Yaskawa INFORM job: X2_55A(90,180).JBI

/JOB
//NAME X2_55A(90,180)
//POS
///NPOS 356,356,356,16,0,0
///TOOL 0
///POSTYPE PULSE
///PULSE
C00000=-1668,-120197,-100216,-7,84052,41
C00001=57589,-42382,-44231,37759,86719,-54272
C00002=65855,-25584,-33137,36767,84603,-51533
C00003=68819,-25314,-30615,36422,82198,-51104
C00004=70004,-25113,-29538,36287,81242,-50929
C00005=71107,-26982,-30843,36133,80649,-50666
C00006=70797,-26613,-30828,36166,80927,-50703
C00007=70799,-26325,-28960,36248,80110,-50973
C00008=70711,-26240,-29288,36240,80345,-50932
C00009=71628,-24021,-27732,36086,80108,-50627
C00010=70711,-26240,-29288,36240,80345,-50932
C00011=69517,-26484,-30393,36372,81303,-51111
C00012=66526,-26862,-32992,36707,83713,-51552
C00013=67184,-38422,-41454,21825,57357,-56847
C00014=69536,-35116,-36433,20931,55446,-56242
C00015=70451,-33735,-34368,20579,54688,-56001
C00016=70453,-33369,-32455,20825,53760,-56193
C00017=71285,-32850,-32302,20328,53712,-55835
C00018=71877,-32425,-32021,19993,53611,-55596
C00019=70458,-33427,-32681,20795,53862,-56169
C00020=69543,-34832,-34766,21144,54620,-56412
C00021=67191,-38201,-39835,22030,56533,-57020
C00022=54852,-62445,-55541,26402,56356,-60471
C00023=66049,-20273,-10630,37753,75560,-54572
C00024=69005,-19201,-7438,37708,73136,-54154
C00025=70188,-18683,-6088,37693,72169,-53986
C00026=71287,-20467,-7387,37603,71596,-53710
C00027=70964,-19947,-7085,37622,71802,-53778
C00028=70966,-19095,-4730,37816,70991,-54071
C00029=70796,-19587,-5250,37820,71120,-54100
C00030=71712,-17458,-3693,37701,70830,-53802
C00031=70796,-19587,-5250,37820,71120,-54100
C00032=66612,-21337,-9914,37854,74525,-54698
C00033=67375,-34871,-26422,23789,50429,-58369
C00034=69718,-31047,-20945,22976,48471,-57749
C00035=70629,-29456,-18687,22656,47689,-57504
C00036=70631,-28720,-16473,23004,46778,-57736
C00037=70516,-28887,-16788,23031,46910,-57759
C00038=71933,-27925,-16136,22175,46608,-57138
C00039=70516,-28887,-16788,23031,46910,-57759
C00040=67258,-34379,-24600,24142,49668,-58622
C00041=57576,-53152,-36186,27516,49078,-61266
C00042=66086,-20118,-10544,37746,75565,-54554
C00043=69039,-19046,-7350,37700,73143,-54137
C00044=70219,-18527,-6000,37685,72176,-53969
C00045=71318,-20312,-7301,37595,71604,-53693
C00046=74451,-19008,-9811,31488,73352,-51630
C00047=71045,-18968,-4611,37811,70952,-54051
C00048=70901,-19378,-5096,37807,71084,-54066
C00049=71814,-17244,-3534,37689,70794,-53769
C00050=70901,-19378,-5096,37807,71084,-54066
C00051=66723,-21136,-9768,37841,74486,-54664
C00052=67447,-34663,-26265,23746,50418,-58339
C00053=69784,-30837,-20782,22936,48460,-57720
C00054=70694,-29244,-18522,22618,47678,-57477
C00055=70696,-28510,-16308,22965,46767,-57708
C00056=70662,-28628,-16633,22933,46904,-57689
C00057=72075,-27660,-15975,22080,46604,-57068
C00058=70662,-28628,-16633,22933,46904,-57689
C00059=67414,-34127,-24457,24044,49660,-58550
C00060=58044,-52471,-35805,27235,49028,-61049
C00061=66074,-20265,-10583,37755,75529,-54572
C00062=69030,-19190,-7387,37710,73105,-54154
C00063=70213,-18669,-6036,37695,72138,-53986
C00064=71313,-20454,-7335,37605,71565,-53710
C00065=76162,-7525,-3808,27332,81993,-47754
C00066=80041,-11320,-7163,21944,78815,-47604
C00067=72377,-20867,-8485,35073,70629,-54310
C00068=73758,-17101,-5731,34844,70264,-53838
C00069=70643,-18935,-5429,37748,71542,-54012
C00070=66856,-20964,-9691,37824,74460,-54615
C00071=67489,-34539,-26167,23723,50410,-58320
C00072=69824,-30709,-20681,22912,48451,-57703
C00073=70732,-29117,-18420,22594,47670,-57460
C00074=70735,-28382,-16205,22941,46757,-57691
C00075=70742,-28505,-16565,22880,46902,-57650
C00076=72154,-27535,-15905,22025,46603,-57029
C00077=70742,-28505,-16565,22880,46902,-57650
C00078=67499,-34008,-24394,23990,49655,-58510
C00079=55453,-57012,-39392,28557,49780,-62094
C00080=66203,-19744,-10147,37744,75471,-54537
C00081=69149,-18659,-6941,37699,73052,-54122
C00082=75064,-17968,-9396,29448,73085,-51466
C00083=75064,-17451,-7778,29552,72447,-51636
C00084=75064,-17968,-9396,29448,73085,-51466
C00085=75946,-19134,-10253,29336,72713,-51212
C00086=75064,-17968,-9396,29448,73085,-51466
C00087=75754,-15898,-7859,29336,72947,-51227
C00088=76424,-13822,-6293,29228,72804,-50997
C00089=75754,-15898,-7859,29336,72947,-51227
C00090=66920,-20695,-9518,37813,74457,-54589
C00091=67621,-34252,-25984,23640,50405,-58260
C00092=69948,-30420,-20490,22831,48447,-57645
C00093=70853,-28824,-18225,22514,47664,-57402
C00094=70856,-28091,-16012,22860,46751,-57633
C00095=70871,-28224,-16368,22798,46887,-57590
C00096=72279,-27249,-15703,21944,46591,-56971
C00097=70871,-28224,-16368,22798,46887,-57590
C00098=67638,-33734,-24209,23906,49640,-58448
C00099=55815,-56530,-39132,28348,49735,-61930
C00100=62040,-49408,-35425,21981,76207,-31792
C00101=60709,-26510,-20047,45346,80057,4684
C00102=66690,-16485,-13360,68369,79312,42512
C00103=69078,-14532,-8904,68579,77025,42081
C00104=70816,-12412,-6652,68580,75744,42186
C00105=70816,-11895,-4924,68755,75432,41836
C00106=70816,-12191,-5902,68656,75607,42033
C00107=71792,-11356,-5257,68617,74964,42180
C00108=70816,-12191,-5902,68656,75607,42033
C00109=66676,-16129,-12001,68472,79065,42229
C00110=63193,-9981,-8398,68470,81776,42168
C00111=63407,-10692,-8959,68465,81623,42187
C00112=66683,-16749,-13563,68371,79313,42507
C00113=69075,-14796,-9109,68581,77024,42076
C00114=70745,-11991,-5797,68649,75667,42041
C00115=70745,-11723,-4902,68740,75507,41860
C00116=70745,-11991,-5797,68649,75667,42041
C00117=71637,-11147,-5144,68611,75079,42177
C00118=70745,-11991,-5797,68649,75667,42041
C00119=66582,-16423,-12216,68478,79121,42207
C00120=63407,-10692,-8959,68465,81623,42187
C00121=63822,-11950,-9936,68455,81327,42223
C00122=66458,-16791,-13600,68382,79463,42478
C00123=68852,-14853,-9158,68587,77174,42046
C00124=70571,-11924,-5724,68657,75780,42012
C00125=70571,-11606,-4670,68763,75592,41800
C00126=70571,-11924,-5724,68657,75780,42012
C00127=71481,-10958,-4978,68619,75184,42152
C00128=70571,-11924,-5724,68657,75780,42012
C00129=66460,-16423,-12212,68483,79202,42190
C00130=63822,-11950,-9936,68455,81327,42223
C00131=63224,-11357,-9448,68476,81731,42145
C00132=66364,-17176,-13856,68391,79512,42447
C00133=68765,-15240,-9419,68598,77218,42018
C00134=70639,-12464,-6107,68665,75719,42002
C00135=70639,-12123,-4981,68778,75517,41775
C00136=70639,-12464,-6107,68665,75719,42002
C00137=71489,-12094,-5823,68633,75155,42124
C00138=70639,-12464,-6107,68665,75719,42002
C00139=66371,-16801,-12525,68486,79261,42177
C00140=63224,-11357,-9448,68476,81731,42145
C00141=61181,-11757,-9356,73697,82866,41546
C00142=64240,-17718,-13856,73666,80649,41737
C00143=66863,-15926,-9805,73862,78342,41311
C00144=68709,-13799,-7108,73949,76887,41250
C00145=68709,-13459,-5991,74053,76732,41018
C00146=68709,-13799,-7108,73949,76887,41250
C00147=69734,-13311,-6738,73933,76180,41366
C00148=68709,-13799,-7108,73949,76887,41250
C00149=64230,-17406,-12625,73747,80472,41470
C00150=61181,-11757,-9356,73697,82866,41546
C00151=66480,6641,10621,68757,84820,39964
C00152=68626,8290,15092,68972,82643,39427
C00153=70241,9673,17100,69092,81355,39410
C00154=70450,6505,14322,69090,81245,39475
C00155=70553,3980,12141,69090,81193,39508
C00156=70814,753,9403,69097,81027,39553
C00157=71023,-1963,7162,69105,80879,39571
C00158=71227,-3841,5652,69116,80729,39580
C00159=71518,-6826,3222,69133,80522,39603
C00160=69728,-7242,2323,68885,80531,50099
C00161=67320,-7984,-1191,68627,82839,50549
C00162=64248,-2156,3507,68551,84943,50186
C00163=64592,9795,13381,68708,86059,39683
C00164=66301,6160,10192,68752,84947,39948
C00165=68453,7795,14646,68964,82767,39414
C00166=70088,9685,17275,69098,81424,39346
C00167=70208,6205,14134,69086,81392,39425
C00168=70495,1625,10245,69093,81174,39488
C00169=70778,-1158,7972,69106,80973,39513
C00170=71096,-3755,5907,69124,80734,39527
C00171=71402,-6742,3472,69143,80510,39552
C00172=69543,-7724,1931,68879,80653,50072
C00173=67128,-8455,-1572,68624,82965,50520
C00174=63402,-1276,4221,68527,85516,50079
C00175=64855,10954,14425,68718,85865,39698
C00176=66657,7118,11039,68762,84696,39982
C00177=68798,8783,15528,68981,82522,39444
C00178=70438,9008,16329,69085,81272,39495
C00179=70615,7069,14708,69094,81154,39519
C00180=70739,4360,12301,69084,81105,39569
C00181=70970,1221,9677,69092,80948,39601
C00182=71176,-1833,7049,69094,80829,39648
C00183=71437,-4529,4843,69103,80644,39673
C00184=71748,-7101,2766,69123,80416,39696
C00185=69913,-6764,2706,68887,80411,50127
C00186=67511,-7518,-820,68629,82715,50578
C00187=63624,-30,5270,68534,85364,50107
C00188=63862,11878,15249,68686,86520,39553
C00189=66390,6402,10413,68754,84881,39955
C00190=68540,8044,14874,68968,82703,39419
C00191=70181,9445,16975,69093,81380,39385
C00192=70335,7584,15341,69094,81297,39426
C00193=70530,3541,11859,69094,81191,39480
C00194=70890,-606,8409,69110,80944,39523
C00195=71179,-3238,6244,69123,80738,39552
C00196=71562,-6771,3374,69142,80464,39582
C00197=69636,-7481,2133,68882,80591,50083
C00198=67224,-8218,-1376,68626,82900,50533
C00199=63822,-1714,3871,68540,85231,50132
C00200=63329,14007,17177,68668,86843,39444
C00201=66569,6880,10830,68760,84758,39974
C00202=68712,8538,15310,68977,82582,39435
C00203=70389,9260,16520,69083,81315,39495
C00204=70547,6829,14451,69087,81218,39527
C00205=70747,3327,11442,69087,81101,39577
C00206=71116,-1091,7744,69098,80857,39626
C00207=71428,-4412,4995,69112,80639,39660
C00208=71772,-7397,2570,69128,80392,39686
C00209=69821,-7002,2515,68886,80471,50113
C00210=67416,-7751,-1005,68628,82777,50563
C00211=63008,846,6000,68515,85778,50026
C00212=63762,-13800,-23397,33384,81143,33846
C00213=63216,-42046,-51440,23378,87636,17578
C00214=45727,-59511,-30756,56000,46415,-83405
C00215=63600,-41118,-24802,45490,45017,-82457
C00216=66225,-37453,-19470,45320,42687,-82205
C00217=66985,-35369,-17022,45296,41990,-82144
C00218=66739,-33567,-15771,45298,42226,-82158
C00219=66552,-32676,-15204,45296,42400,-82170
C00220=66552,-32676,-15204,45296,42400,-82170
C00221=64241,-27257,-11516,47961,46451,-84296
C00222=63989,-25547,-10343,47964,46689,-84302
C00223=63071,-27644,-13011,47925,47562,-84332
C00224=60526,-30752,-18145,47851,49981,-84409
C00225=67770,-16088,-7478,23342,65234,-48964
C00226=70097,-13154,-2242,23053,62997,-48502
C00227=70885,-10205,1160,22956,62242,-48344
C00228=72645,-14691,-2149,21161,60234,-46072
C00229=73604,-17976,-4628,20896,59841,-45756
C00230=73997,-19162,-5529,20787,59690,-45626
C00231=72634,-10889,-524,23061,68772,-42815
C00232=71285,-12419,-2955,23203,69804,-43126
C00233=68920,-15080,-7952,23391,72046,-43578
C00234=69250,-13060,-5710,34890,81335,-68987
C00235=71611,-13509,-3127,34961,78863,-68799
C00236=72615,-13680,-2113,34997,77863,-68700
C00237=73784,-10293,363,34916,77559,-68314
C00238=74145,-9631,950,34900,77394,-68216
C00239=74277,-12968,-24,37387,72337,-67993
C00240=73166,-13154,-1176,37374,73309,-68129
C00241=70646,-13391,-4216,37310,75805,-68335
C00242=64672,-37114,-24557,40064,74903,-69421
C00243=53215,-58476,-44203,47105,47847,-80185
C00244=63376,-45330,-36761,42259,48937,-80324
C00245=66011,-42025,-31781,41802,46642,-79983
C00246=66803,-39374,-28840,41684,45927,-79889
C00247=66435,-37336,-27552,41714,46294,-79914
C00248=66182,-35655,-26450,41719,46557,-79926
C00249=65614,-32529,-24416,41785,47095,-79977
C00250=62864,-31873,-25281,44718,51456,-82098
C00251=60309,-34555,-30014,44934,53856,-82262
C00252=67632,-21338,-34963,21700,78461,-46433
C00253=69966,-19619,-30796,21196,76290,-45976
C00254=70609,-17501,-27911,21077,75486,-45882
C00255=72382,-22586,-31552,19250,73519,-43800
C00256=73091,-25073,-33340,19051,73190,-43592
C00257=73623,-26709,-34473,18903,72933,-43439
C00258=68334,-10665,-22082,28074,86036,-40590
C00259=71158,-18298,-31053,22026,83070,-40626
C00260=68786,-19743,-34997,22436,85266,-41071
C00261=69099,-17947,-30033,34680,91735,-65800
C00262=71464,-19548,-28381,34430,89257,-65615
C00263=72207,-20624,-27936,34359,88268,-65622
C00264=73578,-17057,-25304,34222,87895,-65183
C00265=73664,-17182,-25351,34359,87477,-65108
C00266=73958,-20252,-26156,35949,82486,-64669
C00267=73022,-19832,-26970,36039,83465,-64736
C00268=70499,-18968,-29094,36318,85950,-64959
C00269=63455,-39500,-42592,39134,83172,-66846
C00270=51243,-53894,-27779,53614,43857,-77380
C00271=63855,-40685,-24535,45334,44930,-82346
C00272=66465,-37011,-19188,45164,42603,-82095
C00273=67437,-35339,-16937,45103,41741,-81998
C00274=66941,-33204,-15550,45158,42161,-82061
C00275=66817,-31847,-14581,45135,42294,-82057
C00276=64624,-27572,-11740,47849,46228,-84190
C00277=64311,-26098,-10734,47854,46491,-84221
C00278=64293,-25560,-10405,47823,46547,-84177
C00279=63305,-27217,-12717,47811,47464,-84242
C00280=60770,-30337,-17865,47737,49880,-84318
C00281=67970,-15627,-7133,23286,65199,-48891
C00282=70291,-12681,-1881,22998,62963,-48432
C00283=71307,-8174,3024,22861,62033,-48217
C00284=73187,-13252,-828,21009,60026,-45895
C00285=74131,-16110,-2954,20747,59640,-45582
C00286=74790,-17977,-4358,20564,59385,-45359
C00287=73591,-11134,-229,22389,66343,-43306
C00288=71473,-11939,-2585,23166,69769,-43061
C00289=69116,-14612,-7597,23356,72011,-43511
C00290=69432,-12586,-5379,34880,81293,-68925
C00291=71788,-13028,-2792,34949,78823,-68737
C00292=72964,-11539,-314,34982,77714,-68604
C00293=73550,-9682,1008,34936,77586,-68401
C00294=74749,-6790,3408,35063,76771,-68013
C00295=74665,-10634,1938,37355,72161,-67883
C00296=73339,-12668,-837,37353,73266,-68068
C00297=70826,-12915,-3884,37290,75759,-68273
C00298=65113,-35015,-20365,40278,73539,-69756
C00299=53349,-51371,-26388,52538,42939,-79703
C00300=63472,-41334,-24935,45567,45062,-82513
C00301=66103,-37674,-19610,45398,42729,-82260
C00302=66910,-34858,-16606,45329,42032,-82167
C00303=66599,-33404,-15701,45331,42324,-82187
C00304=66430,-31981,-14703,45315,42495,-82190
C00305=66430,-31981,-14703,45315,42495,-82190
C00306=64006,-26658,-11208,47976,46658,-84316
C00307=63888,-25248,-10138,47982,46761,-84322
C00308=62953,-27859,-13158,47983,47611,-84376
C00309=60402,-30960,-18285,47908,50032,-84454
C00310=67669,-16318,-7651,23369,65251,-49000
C00311=70002,-13390,-2423,23080,63015,-48538
C00312=70899,-10391,1111,22963,62182,-48353
C00313=72647,-15243,-2568,21159,60210,-46076
C00314=73303,-17639,-4445,20974,59974,-45854
C00315=74110,-19941,-6134,20754,59636,-45590
C00316=72493,-11008,-705,23079,68858,-42852
C00317=71192,-12658,-3138,23220,69821,-43159
C00318=68821,-15313,-8129,23409,72064,-43613
C00319=69142,-13291,-5919,34893,81386,-69015
C00320=71506,-13748,-3343,34964,78914,-68825
C00321=72645,-14152,-2445,34999,77819,-68703
C00322=73632,-10983,-133,34929,77580,-68369
C00323=74146,-10154,664,35099,76986,-68198
C00324=74270,-12868,107,37392,72315,-68004
C00325=73063,-13399,-1397,37382,73361,-68153
C00326=70541,-13628,-4430,37317,75858,-68362
C00327=62799,-35833,-17070,40889,72727,-71130
C00328=50528,-54679,-28205,53954,44180,-82418
C00329=63728,-40900,-24669,45411,44974,-82401
C00330=66345,-37233,-19330,45240,42645,-82150
C00331=67222,-34909,-16728,45138,41913,-82032
C00332=66918,-33222,-15549,45178,42162,-82073
C00333=64515,-27645,-11825,47864,46297,-84213
C00334=64210,-25261,-10133,47870,46583,-84229
C00335=63188,-27431,-12864,47868,47513,-84286
C00336=60648,-30543,-18005,47795,49931,-84362
C00337=67871,-15857,-7305,23313,65216,-48928
C00338=70194,-12918,-2061,23025,62980,-48468
C00339=71394,-8811,2530,22846,61988,-48193
C00340=73185,-13936,-1404,21008,60030,-45891
C00341=74121,-17196,-3945,20740,59690,-45575
C00342=74788,-18894,-5176,20558,59417,-45353
C00343=73089,-9260,877,22982,68622,-42667
C00344=71380,-12178,-2769,23185,69787,-43094
C00345=69019,-14846,-7774,23374,72029,-43544
C00346=69337,-12822,-5559,34885,81324,-68954
C00347=71694,-13269,-2976,34955,78854,-68766
C00348=73044,-12528,-1211,34971,77719,-68569
C00349=73788,-10413,417,34925,77477,-68337
C00350=75391,-6243,3707,34832,76922,-67850
C00351=74818,-11558,1118,37336,72118,-67834
C00352=73247,-12912,-1024,37363,73298,-68096
C00353=70733,-13152,-4066,37299,75792,-68302
C00354=61251,-34042,-18878,37994,78635,-71374
C00355=-1877,-120204,-100218,-7,84050,43
BC00000=198907,523889,911617
BC00001=345014,523889,1075139
BC00002=345014,523889,1075139
BC00003=345014,523889,1075139
BC00004=345014,523889,1075139
BC00005=345014,523889,1075139
BC00006=345014,523889,1075139
BC00007=345014,523889,1075139
BC00008=345014,523889,1075139
BC00009=345014,523889,1075139
BC00010=345014,523889,1075139
BC00011=345014,523889,1075139
BC00012=345014,523889,1075139
BC00013=319991,523889,1075139
BC00014=319991,523889,1075139
BC00015=319991,523889,1075139
BC00016=319991,523889,1075139
BC00017=319991,523889,1075139
BC00018=319991,523889,1075139
BC00019=319991,523889,1075139
BC00020=319991,523889,1075139
BC00021=319991,523889,1075139
BC00022=314787,523428,1075139
BC00023=345007,523889,1034671
BC00024=345007,523889,1034671
BC00025=345007,523889,1034671
BC00026=345007,523889,1034671
BC00027=345007,523889,1034671
BC00028=345007,523889,1034671
BC00029=345007,523889,1034671
BC00030=345007,523889,1034671
BC00031=345007,523889,1034671
BC00032=345007,523889,1034671
BC00033=320020,523889,995543
BC00034=320020,523889,995543
BC00035=320020,523889,995543
BC00036=320020,523889,995543
BC00037=320020,523889,995543
BC00038=320020,523889,995543
BC00039=320020,523889,995543
BC00040=320020,523889,995543
BC00041=314822,523428,1004781
BC00042=344944,523889,872722
BC00043=344944,523889,872722
BC00044=344944,523889,872722
BC00045=344944,523889,872722
BC00046=344944,523889,872722
BC00047=344944,523889,872722
BC00048=344944,523889,872722
BC00049=344944,523889,872722
BC00050=344944,523889,872722
BC00051=344944,523889,872722
BC00052=320194,523889,833570
BC00053=320194,523889,833570
BC00054=320194,523889,833570
BC00055=320194,523889,833570
BC00056=320194,523889,833570
BC00057=320194,523889,833570
BC00058=320194,523889,833570
BC00059=320194,523889,833570
BC00060=314856,523428,843479
BC00061=345071,523889,710473
BC00062=345071,523889,710473
BC00063=345071,523889,710473
BC00064=345071,523889,710473
BC00065=345071,523889,710473
BC00066=345071,523889,710473
BC00067=345071,523889,710473
BC00068=345071,523889,710473
BC00069=345071,523889,710473
BC00070=345071,523889,710473
BC00071=320030,523889,671561
BC00072=320030,523889,671561
BC00073=320030,523889,671561
BC00074=320030,523889,671561
BC00075=320030,523889,671561
BC00076=320030,523889,671561
BC00077=320030,523889,671561
BC00078=320030,523889,671561
BC00079=314891,523428,682178
BC00080=344897,523889,548956
BC00081=344897,523889,548956
BC00082=344897,523889,548956
BC00083=344897,523889,548956
BC00084=344897,523889,548956
BC00085=344897,523889,548956
BC00086=344897,523889,548956
BC00087=344897,523889,548956
BC00088=344897,523889,548956
BC00089=344897,523889,548956
BC00090=344897,523889,548956
BC00091=320155,523889,510231
BC00092=320155,523889,510231
BC00093=320155,523889,510231
BC00094=320155,523889,510231
BC00095=320155,523889,510231
BC00096=320155,523889,510231
BC00097=320155,523889,510231
BC00098=320155,523889,510231
BC00099=314926,523428,520876
BC00100=378632,511033,578885
BC00101=388395,517461,490334
BC00102=398158,523889,401783
BC00103=398158,523889,401783
BC00104=398158,523889,401783
BC00105=398158,523889,401783
BC00106=398158,523889,401783
BC00107=398158,523889,401783
BC00108=398158,523889,401783
BC00109=398158,523889,401783
BC00110=398158,523889,401783
BC00111=398158,523889,563053
BC00112=398158,523889,563053
BC00113=398158,523889,563053
BC00114=398158,523889,563053
BC00115=398158,523889,563053
BC00116=398158,523889,563053
BC00117=398158,523889,563053
BC00118=398158,523889,563053
BC00119=398158,523889,563053
BC00120=398158,523889,563053
BC00121=398158,523889,725125
BC00122=398158,523889,725125
BC00123=398158,523889,725125
BC00124=398158,523889,725125
BC00125=398158,523889,725125
BC00126=398158,523889,725125
BC00127=398158,523889,725125
BC00128=398158,523889,725125
BC00129=398158,523889,725125
BC00130=398158,523889,725125
BC00131=398158,523889,887425
BC00132=398158,523889,887425
BC00133=398158,523889,887425
BC00134=398158,523889,887425
BC00135=398158,523889,887425
BC00136=398158,523889,887425
BC00137=398158,523889,887425
BC00138=398158,523889,887425
BC00139=398158,523889,887425
BC00140=398158,523889,887425
BC00141=398158,523889,1018488
BC00142=398158,523889,1018488
BC00143=398158,523889,1018488
BC00144=398158,523889,1018488
BC00145=398158,523889,1018488
BC00146=398158,523889,1018488
BC00147=398158,523889,1018488
BC00148=398158,523889,1018488
BC00149=398158,523889,1018488
BC00150=398158,523889,1018488
BC00151=398158,523889,750776
BC00152=398158,523889,750776
BC00153=398158,523889,750776
BC00154=398158,523889,750776
BC00155=398158,523889,750776
BC00156=398158,523889,750776
BC00157=398158,523889,750776
BC00158=398158,523889,750776
BC00159=398158,523889,750776
BC00160=398158,523889,750776
BC00161=398158,523889,750776
BC00162=398158,523889,750776
BC00163=398158,523889,1074935
BC00164=398158,523889,1074935
BC00165=398158,523889,1074935
BC00166=398158,523889,1074935
BC00167=398158,523889,1074935
BC00168=398158,523889,1074935
BC00169=398158,523889,1074935
BC00170=398158,523889,1074935
BC00171=398158,523889,1074935
BC00172=398158,523889,1074935
BC00173=398158,523889,1074935
BC00174=398158,523889,1074935
BC00175=398158,523889,427370
BC00176=398158,523889,427370
BC00177=398158,523889,427370
BC00178=398158,523889,427370
BC00179=398158,523889,427370
BC00180=398158,523889,427370
BC00181=398158,523889,427370
BC00182=398158,523889,427370
BC00183=398158,523889,427370
BC00184=398158,523889,427370
BC00185=398158,523889,427370
BC00186=398158,523889,427370
BC00187=398158,523889,427370
BC00188=398158,523889,912882
BC00189=398158,523889,912882
BC00190=398158,523889,912882
BC00191=398158,523889,912882
BC00192=398158,523889,912882
BC00193=398158,523889,912882
BC00194=398158,523889,912882
BC00195=398158,523889,912882
BC00196=398158,523889,912882
BC00197=398158,523889,912882
BC00198=398158,523889,912882
BC00199=398158,523889,912882
BC00200=398158,523889,588670
BC00201=398158,523889,588670
BC00202=398158,523889,588670
BC00203=398158,523889,588670
BC00204=398158,523889,588670
BC00205=398158,523889,588670
BC00206=398158,523889,588670
BC00207=398158,523889,588670
BC00208=398158,523889,588670
BC00209=398158,523889,588670
BC00210=398158,523889,588670
BC00211=398158,523889,588670
BC00212=398158,523428,626531
BC00213=360182,523428,720894
BC00214=313344,523428,837276
BC00215=325280,523889,810101
BC00216=325280,523889,810101
BC00217=325280,523889,810101
BC00218=325280,523889,810101
BC00219=325280,523889,810101
BC00220=325280,523889,810101
BC00221=325280,523889,810101
BC00222=325280,523889,810101
BC00223=325280,523889,810101
BC00224=325280,523889,810101
BC00225=319297,523889,902511
BC00226=319297,523889,902511
BC00227=319297,523889,902511
BC00228=319297,523889,902511
BC00229=319297,523889,902511
BC00230=319297,523889,902511
BC00231=319297,523889,902511
BC00232=319297,523889,902511
BC00233=319297,523889,902511
BC00234=349953,523889,883368
BC00235=349953,523889,883368
BC00236=349953,523889,883368
BC00237=349953,523889,883368
BC00238=349953,523889,883368
BC00239=349953,523889,883368
BC00240=349953,523889,883368
BC00241=349953,523889,883368
BC00242=354739,523428,897913
BC00243=313274,523428,1075139
BC00244=325274,523889,1075139
BC00245=325274,523889,1075139
BC00246=325274,523889,1075139
BC00247=325274,523889,1075139
BC00248=325274,523889,1075139
BC00249=325274,523889,1075139
BC00250=325274,523889,1075139
BC00251=325274,523889,1075139
BC00252=319291,523889,1075139
BC00253=319291,523889,1075139
BC00254=319291,523889,1075139
BC00255=319291,523889,1075139
BC00256=319291,523889,1075139
BC00257=319291,523889,1075139
BC00258=319291,523889,1075139
BC00259=319291,523889,1075139
BC00260=319291,523889,1075139
BC00261=349918,523889,1075139
BC00262=349918,523889,1075139
BC00263=349918,523889,1075139
BC00264=349918,523889,1075139
BC00265=349918,523889,1075139
BC00266=349918,523889,1075139
BC00267=349918,523889,1075139
BC00268=349918,523889,1075139
BC00269=354669,523428,1075139
BC00270=313414,523428,513866
BC00271=325287,523889,486695
BC00272=325287,523889,486695
BC00273=325287,523889,486695
BC00274=325287,523889,486695
BC00275=325287,523889,486695
BC00276=325287,523889,486695
BC00277=325287,523889,486695
BC00278=325287,523888,486694
BC00279=325287,523889,486695
BC00280=325287,523889,486695
BC00281=319304,523889,579105
BC00282=319304,523889,579105
BC00283=319304,523889,579105
BC00284=319304,523889,579105
BC00285=319304,523889,579105
BC00286=319304,523889,579105
BC00287=319304,523889,579105
BC00288=319304,523889,579105
BC00289=319304,523889,579105
BC00290=349931,523889,559759
BC00291=349931,523889,559759
BC00292=349931,523889,559759
BC00293=349931,523889,559759
BC00294=349931,523889,559759
BC00295=349931,523889,559759
BC00296=349931,523889,559759
BC00297=349931,523889,559759
BC00298=354809,523428,574503
BC00299=313309,523428,999384
BC00300=325277,523889,972207
BC00301=325277,523889,972207
BC00302=325277,523889,972207
BC00303=325277,523889,972207
BC00304=325277,523889,972207
BC00305=325277,523889,972207
BC00306=325277,523889,972207
BC00307=325277,523889,972207
BC00308=325277,523889,972207
BC00309=325277,523889,972207
BC00310=319294,523889,1064617
BC00311=319294,523889,1064617
BC00312=319294,523889,1064617
BC00313=319294,523889,1064617
BC00314=319294,523889,1064617
BC00315=319294,523889,1064617
BC00316=319294,523889,1064617
BC00317=319294,523889,1064617
BC00318=319294,523889,1064617
BC00319=349921,523889,1045272
BC00320=349921,523889,1045272
BC00321=349921,523889,1045272
BC00322=349921,523889,1045272
BC00323=349921,523889,1045272
BC00324=349921,523889,1045272
BC00325=349921,523889,1045272
BC00326=349921,523889,1045272
BC00327=354704,523428,1060021
BC00328=313379,523428,675168
BC00329=325283,523889,647995
BC00330=325283,523889,647995
BC00331=325283,523889,647995
BC00332=325283,523889,647995
BC00333=325283,523889,647995
BC00334=325283,523889,647995
BC00335=325283,523889,647995
BC00336=325283,523889,647995
BC00337=319300,523889,740405
BC00338=319300,523889,740405
BC00339=319300,523889,740405
BC00340=319300,523889,740405
BC00341=319300,523889,740405
BC00342=319300,523889,740405
BC00343=319300,523889,740405
BC00344=319300,523889,740405
BC00345=319300,523889,740405
BC00346=349928,523889,721059
BC00347=349928,523889,721059
BC00348=349928,523889,721059
BC00349=349928,523889,721059
BC00350=349928,523889,721059
BC00351=349928,523889,721059
BC00352=349928,523889,721059
BC00353=349928,523889,721059
BC00354=349928,523889,721059
BC00355=87745,523889,1075193
EC00000=-798156,-1296783
EC00001=-798156,-1296783
EC00002=-798156,-1296783
EC00003=-798156,-1296783
EC00004=-798156,-1296783
EC00005=-798156,-1296783
EC00006=-798156,-1296783
EC00007=-798156,-1296783
EC00008=-798156,-1296783
EC00009=-798156,-1296783
EC00010=-798156,-1296783
EC00011=-798156,-1296783
EC00012=-798156,-1296783
EC00013=-798156,-1296783
EC00014=-798156,-1296783
EC00015=-798156,-1296783
EC00016=-798156,-1296783
EC00017=-798156,-1296783
EC00018=-798156,-1296783
EC00019=-798156,-1296783
EC00020=-798156,-1296783
EC00021=-798156,-1296783
EC00022=-798156,-1296783
EC00023=-798156,-1296783
EC00024=-798156,-1296783
EC00025=-798156,-1296783
EC00026=-798156,-1296783
EC00027=-798156,-1296783
EC00028=-798156,-1296783
EC00029=-798156,-1296783
EC00030=-798156,-1296783
EC00031=-798156,-1296783
EC00032=-798156,-1296783
EC00033=-798156,-1296783
EC00034=-798156,-1296783
EC00035=-798156,-1296783
EC00036=-798156,-1296783
EC00037=-798156,-1296783
EC00038=-798156,-1296783
EC00039=-798156,-1296783
EC00040=-798156,-1296783
EC00041=-798156,-1296783
EC00042=-798156,-1296783
EC00043=-798156,-1296783
EC00044=-798156,-1296783
EC00045=-798156,-1296783
EC00046=-798156,-1296783
EC00047=-798156,-1296783
EC00048=-798156,-1296783
EC00049=-798156,-1296783
EC00050=-798156,-1296783
EC00051=-798156,-1296783
EC00052=-798156,-1296783
EC00053=-798156,-1296783
EC00054=-798156,-1296783
EC00055=-798156,-1296783
EC00056=-798156,-1296783
EC00057=-798156,-1296783
EC00058=-798156,-1296783
EC00059=-798156,-1296783
EC00060=-798156,-1296783
EC00061=-798156,-1296783
EC00062=-798156,-1296783
EC00063=-798156,-1296783
EC00064=-798156,-1296783
EC00065=-798156,-1296783
EC00066=-798156,-1296783
EC00067=-798156,-1296783
EC00068=-798156,-1296783
EC00069=-798156,-1296783
EC00070=-798156,-1296783
EC00071=-798156,-1296783
EC00072=-798156,-1296783
EC00073=-798156,-1296783
EC00074=-798156,-1296783
EC00075=-798156,-1296783
EC00076=-798156,-1296783
EC00077=-798156,-1296783
EC00078=-798156,-1296783
EC00079=-798156,-1296783
EC00080=-798156,-1296783
EC00081=-798156,-1296783
EC00082=-798156,-1296783
EC00083=-798156,-1296783
EC00084=-798156,-1296783
EC00085=-798156,-1296783
EC00086=-798156,-1296783
EC00087=-798156,-1296783
EC00088=-798156,-1296783
EC00089=-798156,-1296783
EC00090=-798156,-1296783
EC00091=-798156,-1296783
EC00092=-798156,-1296783
EC00093=-798156,-1296783
EC00094=-798156,-1296783
EC00095=-798156,-1296783
EC00096=-798156,-1296783
EC00097=-798156,-1296783
EC00098=-798156,-1296783
EC00099=-798156,-1296783
EC00100=-798156,-1296783
EC00101=-798156,-1296783
EC00102=-798156,-1296783
EC00103=-798156,-1296783
EC00104=-798156,-1296783
EC00105=-798156,-1296783
EC00106=-798156,-1296783
EC00107=-798156,-1296783
EC00108=-798156,-1296783
EC00109=-798156,-1296783
EC00110=-798156,-1296783
EC00111=-798156,-1296783
EC00112=-798156,-1296783
EC00113=-798156,-1296783
EC00114=-798156,-1296783
EC00115=-798156,-1296783
EC00116=-798156,-1296783
EC00117=-798156,-1296783
EC00118=-798156,-1296783
EC00119=-798156,-1296783
EC00120=-798156,-1296783
EC00121=-798156,-1296783
EC00122=-798156,-1296783
EC00123=-798156,-1296783
EC00124=-798156,-1296783
EC00125=-798156,-1296783
EC00126=-798156,-1296783
EC00127=-798156,-1296783
EC00128=-798156,-1296783
EC00129=-798156,-1296783
EC00130=-798156,-1296783
EC00131=-798156,-1296783
EC00132=-798156,-1296783
EC00133=-798156,-1296783
EC00134=-798156,-1296783
EC00135=-798156,-1296783
EC00136=-798156,-1296783
EC00137=-798156,-1296783
EC00138=-798156,-1296783
EC00139=-798156,-1296783
EC00140=-798156,-1296783
EC00141=-798156,-1296783
EC00142=-798156,-1296783
EC00143=-798156,-1296783
EC00144=-798156,-1296783
EC00145=-798156,-1296783
EC00146=-798156,-1296783
EC00147=-798156,-1296783
EC00148=-798156,-1296783
EC00149=-798156,-1296783
EC00150=-798156,-1296783
EC00151=-798156,-1296783
EC00152=-798156,-1296783
EC00153=-798156,-1296783
EC00154=-798156,-1296783
EC00155=-798156,-1296783
EC00156=-798156,-1296783
EC00157=-798156,-1296783
EC00158=-798156,-1296783
EC00159=-798156,-1296783
EC00160=-798156,-1296783
EC00161=-798156,-1296783
EC00162=-798156,-1296783
EC00163=-798156,-1296783
EC00164=-798156,-1296783
EC00165=-798156,-1296783
EC00166=-798156,-1296783
EC00167=-798156,-1296783
EC00168=-798156,-1296783
EC00169=-798156,-1296783
EC00170=-798156,-1296783
EC00171=-798156,-1296783
EC00172=-798156,-1296783
EC00173=-798156,-1296783
EC00174=-798156,-1296783
EC00175=-798156,-1296783
EC00176=-798156,-1296783
EC00177=-798156,-1296783
EC00178=-798156,-1296783
EC00179=-798156,-1296783
EC00180=-798156,-1296783
EC00181=-798156,-1296783
EC00182=-798156,-1296783
EC00183=-798156,-1296783
EC00184=-798156,-1296783
EC00185=-798156,-1296783
EC00186=-798156,-1296783
EC00187=-798156,-1296783
EC00188=-798156,-1296783
EC00189=-798156,-1296783
EC00190=-798156,-1296783
EC00191=-798156,-1296783
EC00192=-798156,-1296783
EC00193=-798156,-1296783
EC00194=-798156,-1296783
EC00195=-798156,-1296783
EC00196=-798156,-1296783
EC00197=-798156,-1296783
EC00198=-798156,-1296783
EC00199=-798156,-1296783
EC00200=-798156,-1296783
EC00201=-798156,-1296783
EC00202=-798156,-1296783
EC00203=-798156,-1296783
EC00204=-798156,-1296783
EC00205=-798156,-1296783
EC00206=-798156,-1296783
EC00207=-798156,-1296783
EC00208=-798156,-1296783
EC00209=-798156,-1296783
EC00210=-798156,-1296783
EC00211=-798156,-1296783
EC00212=-798156,-1296783
EC00213=-798156,-1296783
EC00214=-798156,-1296783
EC00215=-798156,-1296783
EC00216=-798156,-1296783
EC00217=-798156,-1296783
EC00218=-798156,-1296783
EC00219=-798156,-1296783
EC00220=-798156,-1296783
EC00221=-798156,-1296783
EC00222=-798156,-1296783
EC00223=-798156,-1296783
EC00224=-798156,-1296783
EC00225=-798156,-1296783
EC00226=-798156,-1296783
EC00227=-798156,-1296783
EC00228=-798156,-1296783
EC00229=-798156,-1296783
EC00230=-798156,-1296783
EC00231=-798156,-1296783
EC00232=-798156,-1296783
EC00233=-798156,-1296783
EC00234=-798156,-1296783
EC00235=-798156,-1296783
EC00236=-798156,-1296783
EC00237=-798156,-1296783
EC00238=-798156,-1296783
EC00239=-798156,-1296783
EC00240=-798156,-1296783
EC00241=-798156,-1296783
EC00242=-798156,-1296783
EC00243=-798156,-1296783
EC00244=-798156,-1296783
EC00245=-798156,-1296783
EC00246=-798156,-1296783
EC00247=-798156,-1296783
EC00248=-798156,-1296783
EC00249=-798156,-1296783
EC00250=-798156,-1296783
EC00251=-798156,-1296783
EC00252=-798156,-1296783
EC00253=-798156,-1296783
EC00254=-798156,-1296783
EC00255=-798156,-1296783
EC00256=-798156,-1296783
EC00257=-798156,-1296783
EC00258=-798156,-1296783
EC00259=-798156,-1296783
EC00260=-798156,-1296783
EC00261=-798156,-1296783
EC00262=-798156,-1296783
EC00263=-798156,-1296783
EC00264=-798156,-1296783
EC00265=-798156,-1296783
EC00266=-798156,-1296783
EC00267=-798156,-1296783
EC00268=-798156,-1296783
EC00269=-798156,-1296783
EC00270=-798156,-1296783
EC00271=-798156,-1296783
EC00272=-798156,-1296783
EC00273=-798156,-1296783
EC00274=-798156,-1296783
EC00275=-798156,-1296783
EC00276=-798156,-1296783
EC00277=-798156,-1296783
EC00278=-798154,-1296781
EC00279=-798156,-1296783
EC00280=-798156,-1296783
EC00281=-798156,-1296783
EC00282=-798156,-1296783
EC00283=-798156,-1296783
EC00284=-798156,-1296783
EC00285=-798156,-1296783
EC00286=-798156,-1296783
EC00287=-798156,-1296783
EC00288=-798156,-1296783
EC00289=-798156,-1296783
EC00290=-798156,-1296783
EC00291=-798156,-1296783
EC00292=-798156,-1296783
EC00293=-798156,-1296783
EC00294=-798156,-1296783
EC00295=-798156,-1296783
EC00296=-798156,-1296783
EC00297=-798156,-1296783
EC00298=-798156,-1296783
EC00299=-798156,-1296783
EC00300=-798156,-1296783
EC00301=-798156,-1296783
EC00302=-798156,-1296783
EC00303=-798156,-1296783
EC00304=-798156,-1296783
EC00305=-798156,-1296783
EC00306=-798156,-1296783
EC00307=-798156,-1296783
EC00308=-798156,-1296783
EC00309=-798156,-1296783
EC00310=-798156,-1296783
EC00311=-798156,-1296783
EC00312=-798156,-1296783
EC00313=-798156,-1296783
EC00314=-798156,-1296783
EC00315=-798156,-1296783
EC00316=-798156,-1296783
EC00317=-798156,-1296783
EC00318=-798156,-1296783
EC00319=-798156,-1296783
EC00320=-798156,-1296783
EC00321=-798156,-1296783
EC00322=-798156,-1296783
EC00323=-798156,-1296783
EC00324=-798156,-1296783
EC00325=-798156,-1296783
EC00326=-798156,-1296783
EC00327=-798156,-1296783
EC00328=-798156,-1296783
EC00329=-798156,-1296783
EC00330=-798156,-1296783
EC00331=-798156,-1296783
EC00332=-798156,-1296783
EC00333=-798156,-1296783
EC00334=-798156,-1296783
EC00335=-798156,-1296783
EC00336=-798156,-1296783
EC00337=-798156,-1296783
EC00338=-798156,-1296783
EC00339=-798156,-1296783
EC00340=-798156,-1296783
EC00341=-798156,-1296783
EC00342=-798156,-1296783
EC00343=-798156,-1296783
EC00344=-798156,-1296783
EC00345=-798156,-1296783
EC00346=-798156,-1296783
EC00347=-798156,-1296783
EC00348=-798156,-1296783
EC00349=-798156,-1296783
EC00350=-798156,-1296783
EC00351=-798156,-1296783
EC00352=-798156,-1296783
EC00353=-798156,-1296783
EC00354=-798156,-1296783
EC00355=-798156,-1296783
///POSTYPE BASE
///RECTAN
///RCONF 0,0,0,0,1,0,0,0,0,0,0,0,0,0,0,0,0,0,0,0,0,0,0,0
P00006=2.006,1.622,-0.565,0.0000,0.0000,0.0000
P00021=0.073,2.058,-0.109,0.0000,0.0000,0.0000
P00022=2.006,1.622,-0.565,0.0000,0.0000,0.0000
///RCONF 0,0,0,0,0,0,0,0,0,0,0,0,0,0,0,0,0,0,0,0,0,0,0,0
P00023=-2.957,-4.083,2.762,0.0000,0.0000,0.0000
P00031=-0.170,0.039,-0.647,0.0000,0.0000,0.0000
P00032=-0.423,0.157,3.222,0.0000,0.0000,0.0000
P00033=0.854,-1.099,3.047,0.0000,0.0000,0.0000
P00041=-0.109,0.014,0.966,0.0000,0.0000,0.0000
P00042=-0.220,0.371,-0.613,0.0000,0.0000,0.0000
P00043=-0.179,-5.890,-3.227,0.0000,0.0000,0.0000
P00051=-5.945,4.696,-10.293,0.0000,0.0000,0.0000
P00052=-0.153,5.586,-7.982,0.0000,0.0000,0.0000
P00053=0.015,-0.644,-4.942,0.0000,0.0000,0.0000
P00061=1211.499,975.999,-261.374,0.5148,35.2356,175.5099
P00062=1205.574,689.500,-262.704,0.5159,35.2461,175.5270
P00063=1197.217,207.358,-268.729,0.4863,35.2395,175.4586
//INST
///DATE 2024/12/19 12:42
///ATTR SC,RW
///GROUP1 RB1,BS1
///GROUP2 ST1
NOP
'X2_55a(90,180)
MOVJ C00000 BC00000 VJ=100.00  +MOVJ EC00000 VJ=100.00
MOVJ C00001 BC00001 VJ=100.00  +MOVJ EC00001 VJ=100.00
'Path S3757
SFTOF3D
MOVJ C00002 BC00002 VJ=100.00  +MOVJ EC00002 VJ=100.00
MOVL C00003 BC00003 V=800.0  +MOVJ EC00003 VJ=100.00
SMOVL C00004 BC00004 V=166.7  +MOVJ EC00004
SREFP 3 C00005 BC00005  +REFP EC00005
CALL JOB:SEARCH-R1-S13D
SET P021 P006
SFTON3D P021
SMOVL C00006 BC00006 V=166.7  +MOVJ EC00006
SREFP 3 C00007 BC00007  +REFP EC00007
CALL JOB:SEARCH-R1-S13D
SET P021 P006
SFTON3D P021
SMOVL C00008 BC00008 V=166.7  +MOVJ EC00008
SREFP 3 C00009 BC00009  +REFP EC00009
CALL JOB:SEARCH-R1-S13D
SET P021 P006
SFTON3D P021
SMOVL C00010 BC00010 V=166.7  +MOVJ EC00010
MOVL C00011 BC00011 V=800.0  +MOVJ EC00011 VJ=100.00
MOVL C00012 BC00012 V=1000.0  +MOVJ EC00012 VJ=100.00
'EndPath S3757
'Path S3758
SFTOF3D
MOVJ C00013 BC00013 VJ=100.00  +MOVJ EC00013 VJ=100.00
MOVL C00014 BC00014 V=800.0  +MOVJ EC00014 VJ=100.00
SMOVL C00015 BC00015 V=166.7  +MOVJ EC00015
SREFP 3 C00016 BC00016  +REFP EC00016
CALL JOB:SEARCH-R1-S13D
SET P022 P006
SFTON3D P022
SMOVL C00017 BC00017 V=166.7  +MOVJ EC00017
SREFP 3 C00018 BC00018  +REFP EC00018
CALL JOB:SEARCH-R1-S13D
SET P022 P006
SFTON3D P022
SMOVL C00019 BC00019 V=166.7  +MOVJ EC00019
MOVL C00020 BC00020 V=800.0  +MOVJ EC00020 VJ=100.00
MOVL C00021 BC00021 V=1000.0  +MOVJ EC00021 VJ=100.00
'EndPath S3758
MOVJ C00022 BC00022 VJ=100.00  +MOVJ EC00022 VJ=100.00
'
'Path S3759
SFTOF3D
MOVJ C00023 BC00023 VJ=100.00  +MOVJ EC00023 VJ=100.00
MOVL C00024 BC00024 V=800.0  +MOVJ EC00024 VJ=100.00
SMOVL C00025 BC00025 V=166.7  +MOVJ EC00025
SREFP 3 C00026 BC00026  +REFP EC00026
CALL JOB:SEARCH-R1-S13D
SET P031 P006
SFTON3D P031
SMOVL C00027 BC00027 V=166.7  +MOVJ EC00027
SREFP 3 C00028 BC00028  +REFP EC00028
CALL JOB:SEARCH-R1-S13D
SET P031 P006
SFTON3D P031
SMOVL C00029 BC00029 V=166.7  +MOVJ EC00029
SREFP 3 C00030 BC00030  +REFP EC00030
CALL JOB:SEARCH-R1-S13D
SET P031 P006
SFTON3D P031
SMOVL C00031 BC00031 V=166.7  +MOVJ EC00031
MOVL C00032 BC00032 V=1000.0  +MOVJ EC00032 VJ=100.00
'EndPath S3759
'Path S3760
SFTOF3D
MOVJ C00033 BC00033 VJ=100.00  +MOVJ EC00033 VJ=100.00
MOVL C00034 BC00034 V=800.0  +MOVJ EC00034 VJ=100.00
SMOVL C00035 BC00035 V=166.7  +MOVJ EC00035
SREFP 3 C00036 BC00036  +REFP EC00036
CALL JOB:SEARCH-R1-S13D
SET P032 P006
SFTON3D P032
SMOVL C00037 BC00037 V=166.7  +MOVJ EC00037
SREFP 3 C00038 BC00038  +REFP EC00038
CALL JOB:SEARCH-R1-S13D
SET P032 P006
SFTON3D P032
SMOVL C00039 BC00039 V=166.7  +MOVJ EC00039
MOVL C00040 BC00040 V=1000.0  +MOVJ EC00040 VJ=100.00
'EndPath S3760
MOVJ C00041 BC00041 VJ=100.00  +MOVJ EC00041 VJ=100.00
'
'Path S3761
SFTOF3D
MOVJ C00042 BC00042 VJ=100.00  +MOVJ EC00042 VJ=100.00
MOVL C00043 BC00043 V=800.0  +MOVJ EC00043 VJ=100.00
SMOVL C00044 BC00044 V=166.7  +MOVJ EC00044
SREFP 3 C00045 BC00045  +REFP EC00045
CALL JOB:SEARCH-R1-S13D
SET P041 P006
SFTON3D P041
SMOVL C00046 BC00046 V=166.7  +MOVJ EC00046
SREFP 3 C00047 BC00047  +REFP EC00047
CALL JOB:SEARCH-R1-S13D
SET P041 P006
SFTON3D P041
SMOVL C00048 BC00048 V=166.7  +MOVJ EC00048
SREFP 3 C00049 BC00049  +REFP EC00049
CALL JOB:SEARCH-R1-S13D
SET P041 P006
SFTON3D P041
SMOVL C00050 BC00050 V=166.7  +MOVJ EC00050
MOVL C00051 BC00051 V=1000.0  +MOVJ EC00051 VJ=100.00
'EndPath S3761
'Path S3762
SFTOF3D
MOVJ C00052 BC00052 VJ=100.00  +MOVJ EC00052 VJ=100.00
MOVL C00053 BC00053 V=800.0  +MOVJ EC00053 VJ=100.00
SMOVL C00054 BC00054 V=166.7  +MOVJ EC00054
SREFP 3 C00055 BC00055  +REFP EC00055
CALL JOB:SEARCH-R1-S13D
SET P042 P006
SFTON3D P042
SMOVL C00056 BC00056 V=166.7  +MOVJ EC00056
SREFP 3 C00057 BC00057  +REFP EC00057
CALL JOB:SEARCH-R1-S13D
SET P042 P006
SFTON3D P042
SMOVL C00058 BC00058 V=166.7  +MOVJ EC00058
MOVL C00059 BC00059 V=1000.0  +MOVJ EC00059 VJ=100.00
'EndPath S3762
MOVJ C00060 BC00060 VJ=100.00  +MOVJ EC00060 VJ=100.00
'
'Path S3763
SFTOF3D
MOVJ C00061 BC00061 VJ=100.00  +MOVJ EC00061 VJ=100.00
MOVL C00062 BC00062 V=800.0  +MOVJ EC00062 VJ=100.00
SMOVL C00063 BC00063 V=166.7  +MOVJ EC00063
SREFP 3 C00064 BC00064  +REFP EC00064
CALL JOB:SEARCH-R1-S13D
SET P051 P006
SFTON3D P051
SMOVL C00065 BC00065 V=166.7  +MOVJ EC00065
SREFP 3 C00066 BC00066  +REFP EC00066
CALL JOB:SEARCH-R1-S13D
SET P051 P006
SFTON3D P051
SMOVL C00067 BC00067 V=166.7  +MOVJ EC00067
SREFP 3 C00068 BC00068  +REFP EC00068
CALL JOB:SEARCH-R1-S13D
SET P051 P006
SFTON3D P051
SMOVL C00069 BC00069 V=166.7  +MOVJ EC00069
MOVL C00070 BC00070 V=1000.0  +MOVJ EC00070 VJ=100.00
'EndPath S3763
'Path S3764
SFTOF3D
MOVJ C00071 BC00071 VJ=100.00  +MOVJ EC00071 VJ=100.00
MOVL C00072 BC00072 V=800.0  +MOVJ EC00072 VJ=100.00
SMOVL C00073 BC00073 V=166.7  +MOVJ EC00073
SREFP 3 C00074 BC00074  +REFP EC00074
CALL JOB:SEARCH-R1-S13D
SET P052 P006
SFTON3D P052
SMOVL C00075 BC00075 V=166.7  +MOVJ EC00075
SREFP 3 C00076 BC00076  +REFP EC00076
CALL JOB:SEARCH-R1-S13D
SET P052 P006
SFTON3D P052
SMOVL C00077 BC00077 V=166.7  +MOVJ EC00077
MOVL C00078 BC00078 V=1000.0  +MOVJ EC00078 VJ=100.00
'EndPath S3764
MOVJ C00079 BC00079 VJ=100.00  +MOVJ EC00079 VJ=100.00
'
'Path S3765
SFTOF3D
MOVJ C00080 BC00080 VJ=100.00  +MOVJ EC00080 VJ=100.00
MOVL C00081 BC00081 V=800.0  +MOVJ EC00081 VJ=100.00
SMOVL C00082 BC00082 V=166.7  +MOVJ EC00082
SREFP 3 C00083 BC00083  +REFP EC00083
CALL JOB:SEARCH-R1-S13D
SET P061 P006
SFTON3D P061
SMOVL C00084 BC00084 V=166.7  +MOVJ EC00084
SREFP 3 C00085 BC00085  +REFP EC00085
CALL JOB:SEARCH-R1-S13D
SET P061 P006
SFTON3D P061
SMOVL C00086 BC00086 V=166.7  +MOVJ EC00086
SMOVL C00087 BC00087 V=166.7  +MOVJ EC00087
SREFP 3 C00088 BC00088  +REFP EC00088
CALL JOB:SEARCH-R1-S13D
SET P061 P006
SFTON3D P061
SMOVL C00089 BC00089 V=166.7  +MOVJ EC00089
MOVL C00090 BC00090 V=1000.0  +MOVJ EC00090 VJ=100.00
'EndPath S3765
'Path S3766
SFTOF3D
MOVJ C00091 BC00091 VJ=100.00  +MOVJ EC00091 VJ=100.00
MOVL C00092 BC00092 V=800.0  +MOVJ EC00092 VJ=100.00
SMOVL C00093 BC00093 V=166.7  +MOVJ EC00093
SREFP 3 C00094 BC00094  +REFP EC00094
CALL JOB:SEARCH-R1-S13D
SET P062 P006
SFTON3D P062
SMOVL C00095 BC00095 V=166.7  +MOVJ EC00095
SREFP 3 C00096 BC00096  +REFP EC00096
CALL JOB:SEARCH-R1-S13D
SET P062 P006
SFTON3D P062
SMOVL C00097 BC00097 V=166.7  +MOVJ EC00097
MOVL C00098 BC00098 V=1000.0  +MOVJ EC00098 VJ=100.00
'EndPath S3766
MOVJ C00099 BC00099 VJ=100.00  +MOVJ EC00099 VJ=100.00
'
MOVJ C00100 BC00100 VJ=100.00  +MOVJ EC00100 VJ=100.00
MOVJ C00101 BC00101 VJ=100.00  +MOVJ EC00101 VJ=100.00
'Path S3767
SFTOF3D
MOVJ C00102 BC00102 VJ=100.00  +MOVJ EC00102 VJ=100.00
MOVL C00103 BC00103 V=800.0  +MOVJ EC00103 VJ=100.00
SMOVL C00104 BC00104 V=166.7  +MOVJ EC00104
SREFP 3 C00105 BC00105  +REFP EC00105
CALL JOB:SEARCH-R1-S13D
SET P063 P006
SFTON3D P063
SMOVL C00106 BC00106 V=166.7  +MOVJ EC00106
SREFP 3 C00107 BC00107  +REFP EC00107
CALL JOB:SEARCH-R1-S13D
SET P063 P006
SFTON3D P063
SMOVL C00108 BC00108 V=166.7  +MOVJ EC00108
MOVL C00109 BC00109 V=1000.0  +MOVJ EC00109 VJ=100.00
'EndPath S3767
MOVJ C00110 BC00110 VJ=100.00  +MOVJ EC00110 VJ=100.00
MOVJ C00111 BC00111 VJ=100.00  +MOVJ EC00111 VJ=100.00
'Path S3768
SFTOF3D
MOVJ C00112 BC00112 VJ=100.00  +MOVJ EC00112 VJ=100.00
MOVL C00113 BC00113 V=800.0  +MOVJ EC00113 VJ=100.00
SMOVL C00114 BC00114 V=166.7  +MOVJ EC00114
SREFP 3 C00115 BC00115  +REFP EC00115
CALL JOB:SEARCH-R1-S13D
SET P053 P006
SFTON3D P053
SMOVL C00116 BC00116 V=166.7  +MOVJ EC00116
SREFP 3 C00117 BC00117  +REFP EC00117
CALL JOB:SEARCH-R1-S13D
SET P053 P006
SFTON3D P053
SMOVL C00118 BC00118 V=166.7  +MOVJ EC00118
MOVL C00119 BC00119 V=1000.0  +MOVJ EC00119 VJ=100.00
'EndPath S3768
MOVJ C00120 BC00120 VJ=100.00  +MOVJ EC00120 VJ=100.00
MOVJ C00121 BC00121 VJ=100.00  +MOVJ EC00121 VJ=100.00
'Path S3769
SFTOF3D
MOVJ C00122 BC00122 VJ=100.00  +MOVJ EC00122 VJ=100.00
MOVL C00123 BC00123 V=800.0  +MOVJ EC00123 VJ=100.00
SMOVL C00124 BC00124 V=166.7  +MOVJ EC00124
SREFP 3 C00125 BC00125  +REFP EC00125
CALL JOB:SEARCH-R1-S13D
SET P043 P006
SFTON3D P043
SMOVL C00126 BC00126 V=166.7  +MOVJ EC00126
SREFP 3 C00127 BC00127  +REFP EC00127
CALL JOB:SEARCH-R1-S13D
SET P043 P006
SFTON3D P043
SMOVL C00128 BC00128 V=166.7  +MOVJ EC00128
MOVL C00129 BC00129 V=1000.0  +MOVJ EC00129 VJ=100.00
'EndPath S3769
MOVJ C00130 BC00130 VJ=100.00  +MOVJ EC00130 VJ=100.00
MOVJ C00131 BC00131 VJ=100.00  +MOVJ EC00131 VJ=100.00
'Path S3770
SFTOF3D
MOVJ C00132 BC00132 VJ=100.00  +MOVJ EC00132 VJ=100.00
MOVL C00133 BC00133 V=800.0  +MOVJ EC00133 VJ=100.00
SMOVL C00134 BC00134 V=166.7  +MOVJ EC00134
SREFP 3 C00135 BC00135  +REFP EC00135
CALL JOB:SEARCH-R1-S13D
SET P033 P006
SFTON3D P033
SMOVL C00136 BC00136 V=166.7  +MOVJ EC00136
SREFP 3 C00137 BC00137  +REFP EC00137
CALL JOB:SEARCH-R1-S13D
SET P033 P006
SFTON3D P033
SMOVL C00138 BC00138 V=166.7  +MOVJ EC00138
MOVL C00139 BC00139 V=1000.0  +MOVJ EC00139 VJ=100.00
'EndPath S3770
MOVJ C00140 BC00140 VJ=100.00  +MOVJ EC00140 VJ=100.00
MOVJ C00141 BC00141 VJ=100.00  +MOVJ EC00141 VJ=100.00
'Path S3771
SFTOF3D
MOVJ C00142 BC00142 VJ=100.00  +MOVJ EC00142 VJ=100.00
MOVL C00143 BC00143 V=800.0  +MOVJ EC00143 VJ=100.00
SMOVL C00144 BC00144 V=166.7  +MOVJ EC00144
SREFP 3 C00145 BC00145  +REFP EC00145
CALL JOB:SEARCH-R1-S13D
SET P023 P006
SFTON3D P023
SMOVL C00146 BC00146 V=166.7  +MOVJ EC00146
SREFP 3 C00147 BC00147  +REFP EC00147
CALL JOB:SEARCH-R1-S13D
SET P023 P006
SFTON3D P023
SMOVL C00148 BC00148 V=166.7  +MOVJ EC00148
MOVL C00149 BC00149 V=1000.0  +MOVJ EC00149 VJ=100.00
'EndPath S3771
MOVJ C00150 BC00150 VJ=100.00  +MOVJ EC00150 VJ=100.00
'
'
'
'Path W3772
SFTOF3D
SFTON3D P043
MOVJ C00151 BC00151 VJ=100.00  +MOVJ EC00151 VJ=100.00
SMOVL C00152 BC00152 V=800.0  +MOVJ EC00152
SMOVL C00153 BC00153 V=166.7 PL=0  +MOVJ EC00153
MACRO1 MJ#(0) ARGF9
ARCON
SMOVL C00154 BC00154 V=10.0  +MOVJ EC00154
SMOVL C00155 BC00155 V=10.0  +MOVJ EC00155
SMOVL C00156 BC00156 V=10.0  +MOVJ EC00156
SMOVL C00157 BC00157 V=10.0  +MOVJ EC00157
SMOVL C00158 BC00158 V=10.0  +MOVJ EC00158
SMOVL C00159 BC00159 V=10.0  +MOVJ EC00159
ARCOF
SMOVL C00160 BC00160 V=800.0  +MOVJ EC00160
SMOVL C00161 BC00161 V=1000.0  +MOVJ EC00161
SFTOF3D
'EndPath W3772
MOVJ C00162 BC00162 VJ=100.00  +MOVJ EC00162 VJ=100.00
MOVJ C00163 BC00163 VJ=100.00  +MOVJ EC00163 VJ=100.00
'Path W3773
SFTOF3D
SFTON3D P023
MOVJ C00164 BC00164 VJ=100.00  +MOVJ EC00164 VJ=100.00
SMOVL C00165 BC00165 V=800.0  +MOVJ EC00165
SMOVL C00166 BC00166 V=166.7 PL=0  +MOVJ EC00166
ARCON
SMOVL C00167 BC00167 V=10.0  +MOVJ EC00167
SMOVL C00168 BC00168 V=10.0  +MOVJ EC00168
SMOVL C00169 BC00169 V=10.0  +MOVJ EC00169
SMOVL C00170 BC00170 V=10.0  +MOVJ EC00170
SMOVL C00171 BC00171 V=10.0  +MOVJ EC00171
ARCOF
SMOVL C00172 BC00172 V=800.0  +MOVJ EC00172
SMOVL C00173 BC00173 V=1000.0  +MOVJ EC00173
SFTOF3D
'EndPath W3773
MOVJ C00174 BC00174 VJ=100.00  +MOVJ EC00174 VJ=100.00
MOVJ C00175 BC00175 VJ=100.00  +MOVJ EC00175 VJ=100.00
'Path W3774
SFTOF3D
SFTON3D P063
MOVJ C00176 BC00176 VJ=100.00  +MOVJ EC00176 VJ=100.00
SMOVL C00177 BC00177 V=800.0  +MOVJ EC00177
SMOVL C00178 BC00178 V=166.7 PL=0  +MOVJ EC00178
ARCON
SMOVL C00179 BC00179 V=10.0  +MOVJ EC00179
SMOVL C00180 BC00180 V=10.0  +MOVJ EC00180
SMOVL C00181 BC00181 V=10.0  +MOVJ EC00181
SMOVL C00182 BC00182 V=10.0  +MOVJ EC00182
SMOVL C00183 BC00183 V=10.0  +MOVJ EC00183
SMOVL C00184 BC00184 V=10.0  +MOVJ EC00184
ARCOF
SMOVL C00185 BC00185 V=800.0  +MOVJ EC00185
SMOVL C00186 BC00186 V=1000.0  +MOVJ EC00186
SFTOF3D
'EndPath W3774
MOVJ C00187 BC00187 VJ=100.00  +MOVJ EC00187 VJ=100.00
MOVJ C00188 BC00188 VJ=100.00  +MOVJ EC00188 VJ=100.00
'Path W3775
SFTOF3D
SFTON3D P033
MOVJ C00189 BC00189 VJ=100.00  +MOVJ EC00189 VJ=100.00
SMOVL C00190 BC00190 V=800.0  +MOVJ EC00190
SMOVL C00191 BC00191 V=166.7 PL=0  +MOVJ EC00191
ARCON
SMOVL C00192 BC00192 V=10.0  +MOVJ EC00192
SMOVL C00193 BC00193 V=10.0  +MOVJ EC00193
SMOVL C00194 BC00194 V=10.0  +MOVJ EC00194
SMOVL C00195 BC00195 V=10.0  +MOVJ EC00195
SMOVL C00196 BC00196 V=10.0  +MOVJ EC00196
ARCOF
SMOVL C00197 BC00197 V=800.0  +MOVJ EC00197
SMOVL C00198 BC00198 V=1000.0  +MOVJ EC00198
SFTOF3D
'EndPath W3775
MOVJ C00199 BC00199 VJ=100.00  +MOVJ EC00199 VJ=100.00
MOVJ C00200 BC00200 VJ=100.00  +MOVJ EC00200 VJ=100.00
'Path W3776
SFTOF3D
SFTON3D P053
MOVJ C00201 BC00201 VJ=100.00  +MOVJ EC00201 VJ=100.00
SMOVL C00202 BC00202 V=800.0  +MOVJ EC00202
SMOVL C00203 BC00203 V=166.7 PL=0  +MOVJ EC00203
ARCON
SMOVL C00204 BC00204 V=10.0  +MOVJ EC00204
SMOVL C00205 BC00205 V=10.0  +MOVJ EC00205
SMOVL C00206 BC00206 V=10.0  +MOVJ EC00206
SMOVL C00207 BC00207 V=10.0  +MOVJ EC00207
SMOVL C00208 BC00208 V=10.0  +MOVJ EC00208
ARCOF
SMOVL C00209 BC00209 V=800.0  +MOVJ EC00209
SMOVL C00210 BC00210 V=1000.0  +MOVJ EC00210
SFTOF3D
'EndPath W3776
MOVJ C00211 BC00211 VJ=100.00  +MOVJ EC00211 VJ=100.00
MOVJ C00212 BC00212 VJ=100.00  +MOVJ EC00212 VJ=100.00
MOVJ C00213 BC00213 VJ=100.00  +MOVJ EC00213 VJ=100.00
'
MOVJ C00214 BC00214 VJ=100.00  +MOVJ EC00214 VJ=100.00
'Path W3777
SFTOF3D
SFTON3D P042
MOVJ C00215 BC00215 VJ=100.00  +MOVJ EC00215 VJ=100.00
SMOVL C00216 BC00216 V=800.0  +MOVJ EC00216
SMOVL C00217 BC00217 V=166.7 PL=0  +MOVJ EC00217
ARCON
SMOVL C00218 BC00218 V=10.0  +MOVJ EC00218
SMOVL C00219 BC00219 V=10.0  +MOVJ EC00219
SMOVL C00220 BC00220 V=10.0  +MOVJ EC00220
SMOVL C00221 BC00221 V=10.0  +MOVJ EC00221
SMOVL C00222 BC00222 V=10.0  +MOVJ EC00222
ARCOF
SMOVL C00223 BC00223 V=800.0  +MOVJ EC00223
SMOVL C00224 BC00224 V=1000.0  +MOVJ EC00224
SFTOF3D
'EndPath W3777
'Path W3778
SFTOF3D
SFTON3D P041
MOVJ C00225 BC00225 VJ=100.00  +MOVJ EC00225 VJ=100.00
SMOVL C00226 BC00226 V=800.0  +MOVJ EC00226
SMOVL C00227 BC00227 V=166.7 PL=0  +MOVJ EC00227
ARCON
SMOVL C00228 BC00228 V=10.0  +MOVJ EC00228
SMOVL C00229 BC00229 V=10.0  +MOVJ EC00229
SMOVL C00230 BC00230 V=10.0  +MOVJ EC00230
SMOVL C00231 BC00231 V=10.0  +MOVJ EC00231
ARCOF
SMOVL C00232 BC00232 V=800.0  +MOVJ EC00232
SMOVL C00233 BC00233 V=1000.0  +MOVJ EC00233
SFTOF3D
'EndPath W3778
'Path W3779
SFTOF3D
SFTON3D P041
MOVJ C00234 BC00234 VJ=100.00  +MOVJ EC00234 VJ=100.00
SMOVL C00235 BC00235 V=800.0  +MOVJ EC00235
SMOVL C00236 BC00236 V=166.7 PL=0  +MOVJ EC00236
ARCON
SMOVL C00237 BC00237 V=10.0  +MOVJ EC00237
SMOVL C00238 BC00238 V=10.0  +MOVJ EC00238
SMOVL C00239 BC00239 V=10.0  +MOVJ EC00239
ARCOF
SMOVL C00240 BC00240 V=800.0  +MOVJ EC00240
SMOVL C00241 BC00241 V=1000.0  +MOVJ EC00241
SFTOF3D
'EndPath W3779
MOVJ C00242 BC00242 VJ=100.00  +MOVJ EC00242 VJ=100.00
'
'
MOVJ C00243 BC00243 VJ=100.00  +MOVJ EC00243 VJ=100.00
'Path W3780
SFTOF3D
SFTON3D P022
MOVJ C00244 BC00244 VJ=100.00  +MOVJ EC00244 VJ=100.00
SMOVL C00245 BC00245 V=800.0  +MOVJ EC00245
SMOVL C00246 BC00246 V=166.7 PL=0  +MOVJ EC00246
ARCON
SMOVL C00247 BC00247 V=10.0  +MOVJ EC00247
SMOVL C00248 BC00248 V=10.0  +MOVJ EC00248
SMOVL C00249 BC00249 V=10.0  +MOVJ EC00249
ARCOF
SMOVL C00250 BC00250 V=800.0  +MOVJ EC00250
SMOVL C00251 BC00251 V=1000.0  +MOVJ EC00251
SFTOF3D
'EndPath W3780
'Path W3781
SFTOF3D
SFTON3D P021
MOVJ C00252 BC00252 VJ=100.00  +MOVJ EC00252 VJ=100.00
SMOVL C00253 BC00253 V=800.0  +MOVJ EC00253
SMOVL C00254 BC00254 V=166.7 PL=0  +MOVJ EC00254
ARCON
SMOVL C00255 BC00255 V=10.0  +MOVJ EC00255
SMOVL C00256 BC00256 V=10.0  +MOVJ EC00256
SMOVL C00257 BC00257 V=10.0  +MOVJ EC00257
SMOVL C00258 BC00258 V=10.0  +MOVJ EC00258
ARCOF
SMOVL C00259 BC00259 V=800.0  +MOVJ EC00259
SMOVL C00260 BC00260 V=1000.0  +MOVJ EC00260
SFTOF3D
'EndPath W3781
'Path W3782
SFTOF3D
SFTON3D P021
MOVJ C00261 BC00261 VJ=100.00  +MOVJ EC00261 VJ=100.00
SMOVL C00262 BC00262 V=800.0  +MOVJ EC00262
SMOVL C00263 BC00263 V=166.7 PL=0  +MOVJ EC00263
ARCON
SMOVL C00264 BC00264 V=10.0  +MOVJ EC00264
SMOVL C00265 BC00265 V=10.0  +MOVJ EC00265
SMOVL C00266 BC00266 V=10.0  +MOVJ EC00266
ARCOF
SMOVL C00267 BC00267 V=800.0  +MOVJ EC00267
SMOVL C00268 BC00268 V=1000.0  +MOVJ EC00268
SFTOF3D
'EndPath W3782
MOVJ C00269 BC00269 VJ=100.00  +MOVJ EC00269 VJ=100.00
'
'
MOVJ C00270 BC00270 VJ=100.00  +MOVJ EC00270 VJ=100.00
'Path W3783
SFTOF3D
SFTON3D P062
MOVJ C00271 BC00271 VJ=100.00  +MOVJ EC00271 VJ=100.00
SMOVL C00272 BC00272 V=800.0  +MOVJ EC00272
SMOVL C00273 BC00273 V=166.7 PL=0  +MOVJ EC00273
ARCON
SMOVL C00274 BC00274 V=10.0  +MOVJ EC00274
SMOVL C00275 BC00275 V=10.0  +MOVJ EC00275
SMOVL C00276 BC00276 V=10.0  +MOVJ EC00276
SMOVL C00277 BC00277 V=10.0  +MOVJ EC00277
SMOVL C00278 BC00278 V=10.0  +MOVJ EC00278
ARCOF
SMOVL C00279 BC00279 V=800.0  +MOVJ EC00279
SMOVL C00280 BC00280 V=1000.0  +MOVJ EC00280
SFTOF3D
'EndPath W3783
'Path W3784
SFTOF3D
SFTON3D P061
MOVJ C00281 BC00281 VJ=100.00  +MOVJ EC00281 VJ=100.00
SMOVL C00282 BC00282 V=800.0  +MOVJ EC00282
SMOVL C00283 BC00283 V=166.7 PL=0  +MOVJ EC00283
ARCON
SMOVL C00284 BC00284 V=10.0  +MOVJ EC00284
SMOVL C00285 BC00285 V=10.0  +MOVJ EC00285
SMOVL C00286 BC00286 V=10.0  +MOVJ EC00286
SMOVL C00287 BC00287 V=10.0  +MOVJ EC00287
ARCOF
SMOVL C00288 BC00288 V=800.0  +MOVJ EC00288
SMOVL C00289 BC00289 V=1000.0  +MOVJ EC00289
SFTOF3D
'EndPath W3784
'Path W3785
SFTOF3D
SFTON3D P061
MOVJ C00290 BC00290 VJ=100.00  +MOVJ EC00290 VJ=100.00
SMOVL C00291 BC00291 V=800.0  +MOVJ EC00291
SMOVL C00292 BC00292 V=166.7 PL=0  +MOVJ EC00292
ARCON
SMOVL C00293 BC00293 V=10.0  +MOVJ EC00293
SMOVL C00294 BC00294 V=10.0  +MOVJ EC00294
SMOVL C00295 BC00295 V=10.0  +MOVJ EC00295
ARCOF
SMOVL C00296 BC00296 V=800.0  +MOVJ EC00296
SMOVL C00297 BC00297 V=1000.0  +MOVJ EC00297
SFTOF3D
'EndPath W3785
MOVJ C00298 BC00298 VJ=100.00  +MOVJ EC00298 VJ=100.00
'
'
MOVJ C00299 BC00299 VJ=100.00  +MOVJ EC00299 VJ=100.00
'Path W3786
SFTOF3D
SFTON3D P032
MOVJ C00300 BC00300 VJ=100.00  +MOVJ EC00300 VJ=100.00
SMOVL C00301 BC00301 V=800.0  +MOVJ EC00301
SMOVL C00302 BC00302 V=166.7 PL=0  +MOVJ EC00302
ARCON
SMOVL C00303 BC00303 V=10.0  +MOVJ EC00303
SMOVL C00304 BC00304 V=10.0  +MOVJ EC00304
SMOVL C00305 BC00305 V=10.0  +MOVJ EC00305
SMOVL C00306 BC00306 V=10.0  +MOVJ EC00306
SMOVL C00307 BC00307 V=10.0  +MOVJ EC00307
ARCOF
SMOVL C00308 BC00308 V=800.0  +MOVJ EC00308
SMOVL C00309 BC00309 V=1000.0  +MOVJ EC00309
SFTOF3D
'EndPath W3786
'Path W3787
SFTOF3D
SFTON3D P031
MOVJ C00310 BC00310 VJ=100.00  +MOVJ EC00310 VJ=100.00
SMOVL C00311 BC00311 V=800.0  +MOVJ EC00311
SMOVL C00312 BC00312 V=166.7 PL=0  +MOVJ EC00312
ARCON
SMOVL C00313 BC00313 V=10.0  +MOVJ EC00313
SMOVL C00314 BC00314 V=10.0  +MOVJ EC00314
SMOVL C00315 BC00315 V=10.0  +MOVJ EC00315
SMOVL C00316 BC00316 V=10.0  +MOVJ EC00316
ARCOF
SMOVL C00317 BC00317 V=800.0  +MOVJ EC00317
SMOVL C00318 BC00318 V=1000.0  +MOVJ EC00318
SFTOF3D
'EndPath W3787
'Path W3788
SFTOF3D
SFTON3D P031
MOVJ C00319 BC00319 VJ=100.00  +MOVJ EC00319 VJ=100.00
SMOVL C00320 BC00320 V=800.0  +MOVJ EC00320
SMOVL C00321 BC00321 V=166.7 PL=0  +MOVJ EC00321
ARCON
SMOVL C00322 BC00322 V=10.0  +MOVJ EC00322
SMOVL C00323 BC00323 V=10.0  +MOVJ EC00323
SMOVL C00324 BC00324 V=10.0  +MOVJ EC00324
ARCOF
SMOVL C00325 BC00325 V=800.0  +MOVJ EC00325
SMOVL C00326 BC00326 V=1000.0  +MOVJ EC00326
SFTOF3D
'EndPath W3788
MOVJ C00327 BC00327 VJ=100.00  +MOVJ EC00327 VJ=100.00
'
'
MOVJ C00328 BC00328 VJ=100.00  +MOVJ EC00328 VJ=100.00
'Path W3789
SFTOF3D
SFTON3D P052
MOVJ C00329 BC00329 VJ=100.00  +MOVJ EC00329 VJ=100.00
SMOVL C00330 BC00330 V=800.0  +MOVJ EC00330
SMOVL C00331 BC00331 V=166.7 PL=0  +MOVJ EC00331
ARCON
SMOVL C00332 BC00332 V=10.0  +MOVJ EC00332
SMOVL C00333 BC00333 V=10.0  +MOVJ EC00333
SMOVL C00334 BC00334 V=10.0  +MOVJ EC00334
ARCOF
SMOVL C00335 BC00335 V=800.0  +MOVJ EC00335
SMOVL C00336 BC00336 V=1000.0  +MOVJ EC00336
SFTOF3D
'EndPath W3789
'Path W3790
SFTOF3D
SFTON3D P051
MOVJ C00337 BC00337 VJ=100.00  +MOVJ EC00337 VJ=100.00
SMOVL C00338 BC00338 V=800.0  +MOVJ EC00338
SMOVL C00339 BC00339 V=166.7 PL=0  +MOVJ EC00339
ARCON
SMOVL C00340 BC00340 V=10.0  +MOVJ EC00340
SMOVL C00341 BC00341 V=10.0  +MOVJ EC00341
SMOVL C00342 BC00342 V=10.0  +MOVJ EC00342
SMOVL C00343 BC00343 V=10.0  +MOVJ EC00343
ARCOF
SMOVL C00344 BC00344 V=800.0  +MOVJ EC00344
SMOVL C00345 BC00345 V=1000.0  +MOVJ EC00345
SFTOF3D
'EndPath W3790
'Path W3791
SFTOF3D
SFTON3D P051
MOVJ C00346 BC00346 VJ=100.00  +MOVJ EC00346 VJ=100.00
SMOVL C00347 BC00347 V=800.0  +MOVJ EC00347
SMOVL C00348 BC00348 V=166.7 PL=0  +MOVJ EC00348
ARCON
SMOVL C00349 BC00349 V=10.0  +MOVJ EC00349
SMOVL C00350 BC00350 V=10.0  +MOVJ EC00350
SMOVL C00351 BC00351 V=10.0  +MOVJ EC00351
ARCOF
SMOVL C00352 BC00352 V=800.0  +MOVJ EC00352
SMOVL C00353 BC00353 V=1000.0  +MOVJ EC00353
SFTOF3D
'EndPath W3791
MOVJ C00354 BC00354 VJ=100.00  +MOVJ EC00354 VJ=100.00
'
MOVJ C00355 BC00355 VJ=100.00  +MOVJ EC00355 VJ=100.00
END
